Fanuc KAREL source: kb00175.KL

PROGRAM KB00175
%NOLOCKGROUP
%ENVIRONMENT IOSETUP
VAR
P1:INTEGER;P2:INTEGER;P3:INTEGER;P4:INTEGER
BEGIN
--
--
--
P1=1
P2=1
P3=1
P4=1
SET_PORT_VAL(P1,P2,P3,P4)
END KB00175
